(* PLC project Tc2_Standard.LTON Demo, tc3-libraries-kb TwinCAT 3.1 *)
(* stored: creationDateTime 2026-05-10T08:00:00, modificationDateTime 2026-05-10T08:00:00 *)

PROGRAM P_Demo_LTON
  VAR
    fbLTON : LTON;  (* Timer (LTIME) 实例 *)
    bRawIn : BOOL;  (* 原始输入（可能抖动） *)
    bStable : BOOL;  (* 稳定后输出 *)
    ltElapsed : LTIME;  (* 已稳定时间 *)
  END_VAR

            // ============================================================
// Tc2_Standard.LTON 演示程序
// ============================================================
// 场景：高频脉冲计数器消抖：信号稳定 50 μs 后才认为有效
// 验证步骤：
//   1. 把本 PROGRAM 加到 PlcTask 调用列表
//   2. 编译并登录目标
//   1. bRawIn 持续 TRUE 满 50 μs → bStable = TRUE
//   2. bRawIn 中途变 FALSE → ltElapsed 立刻归零，bStable 保持 FALSE
// ============================================================

fbLTON(
    IN := bRawIn,
    PT := LTIME#50US,
    Q  => bStable,
    ET => ltElapsed
);

          
END_PROGRAM
